(* Logix 5000 project; controller cal1632 1756-L62 rev 16.20; software revision 16.05; part 23 of 57 *)
(* tags used below, declared in another part *)
   FAULT : BOOL;
   HMI : BOOL;
   p01r09_pb_global_reset : BOOL;
   p19_ai_prs : REAL;
   p19_ai_tc01 : REAL;
   p19_ao_cv : REAL;
   p19_di_tc01_bo : BOOL;
   p19_di_tc02_bo : BOOL;
   p19_dint_to_hmi : DINT[16];
   p19_do_pump : BOOL;
   p19_param_pid2_ff : REAL;
   p19_param_pid2_kd : REAL;
   p19_param_pid2_ki : REAL;
   p19_param_pid2_kp : REAL;
   p19_param_tc01_dev : REAL;
   p19_param_tc01z : REAL;
   p19_param_tc02z : REAL;
   p19_param_zone_pressure : REAL;
   p19_real_to_hmi : REAL[80];
   p19r05 : routine;
   p19r05_timer_fault : TIMER[4];
   p19r05_timer_warning : TIMER[4];
   p19r06 : routine;
   p19r06_timer_fault : TIMER[4];
   p19r06_timer_warning : TIMER[4];
   p19r07 : routine;
   p19r07_timer_fault : TIMER[4];
   p19r07_timer_warning : TIMER[4];
   p19r30 : routine;
   p19r30_cv_man_sp : REAL;
   p19r30_pid_temp : PID;
   p19r30_pid_temp_pv : DINT;
   p19r30_request_cool : BOOL;
   p19r30_request_manual : BOOL;
   p19r31 : routine;
   p19r31_request_auto_run : BOOL;
(* P19_Advanced_Cooling, continued *)

ROUTINE R05_Dint_to_HMI   (* ladder *)
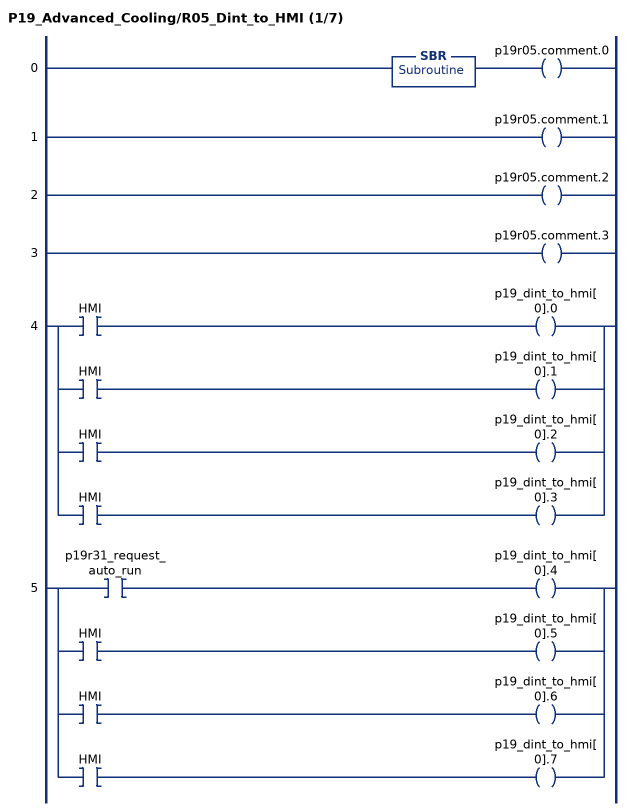
   0: SBR()OTE(p19r05.comment.0);
   1: OTE(p19r05.comment.1);
   2: OTE(p19r05.comment.2);
   3: OTE(p19r05.comment.3);
   4: [XIC(HMI) OTE(p19_dint_to_hmi[0].0) ,XIC(HMI) OTE(p19_dint_to_hmi[0].1) ,XIC(HMI) OTE(p19_dint_to_hmi[0].2) ,XIC(HMI) OTE(p19_dint_to_hmi[0].3) ];
   5: [XIC(p19r31_request_auto_run) OTE(p19_dint_to_hmi[0].4) ,XIC(HMI) OTE(p19_dint_to_hmi[0].5) ,XIC(HMI) OTE(p19_dint_to_hmi[0].6) ,XIC(HMI) OTE(p19_dint_to_hmi[0].7) ];
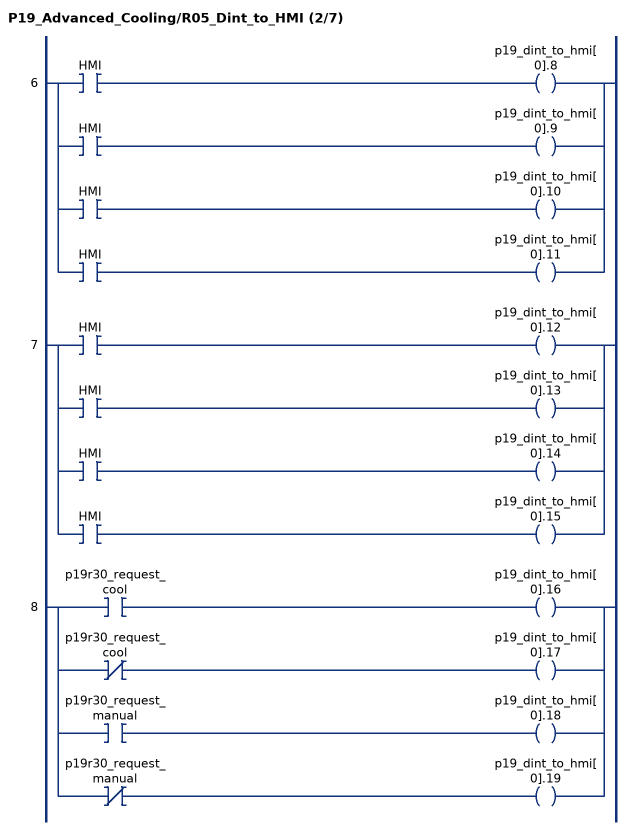
   6: [XIC(HMI) OTE(p19_dint_to_hmi[0].8) ,XIC(HMI) OTE(p19_dint_to_hmi[0].9) ,XIC(HMI) OTE(p19_dint_to_hmi[0].10) ,XIC(HMI) OTE(p19_dint_to_hmi[0].11) ];
   7: [XIC(HMI) OTE(p19_dint_to_hmi[0].12) ,XIC(HMI) OTE(p19_dint_to_hmi[0].13) ,XIC(HMI) OTE(p19_dint_to_hmi[0].14) ,XIC(HMI) OTE(p19_dint_to_hmi[0].15) ];
   8: [XIC(p19r30_request_cool) OTE(p19_dint_to_hmi[0].16) ,XIO(p19r30_request_cool) OTE(p19_dint_to_hmi[0].17) ,XIC(p19r30_request_manual) OTE(p19_dint_to_hmi[0].18) ,XIO(p19r30_request_manual) OTE(p19_dint_to_hmi[0].19) ];
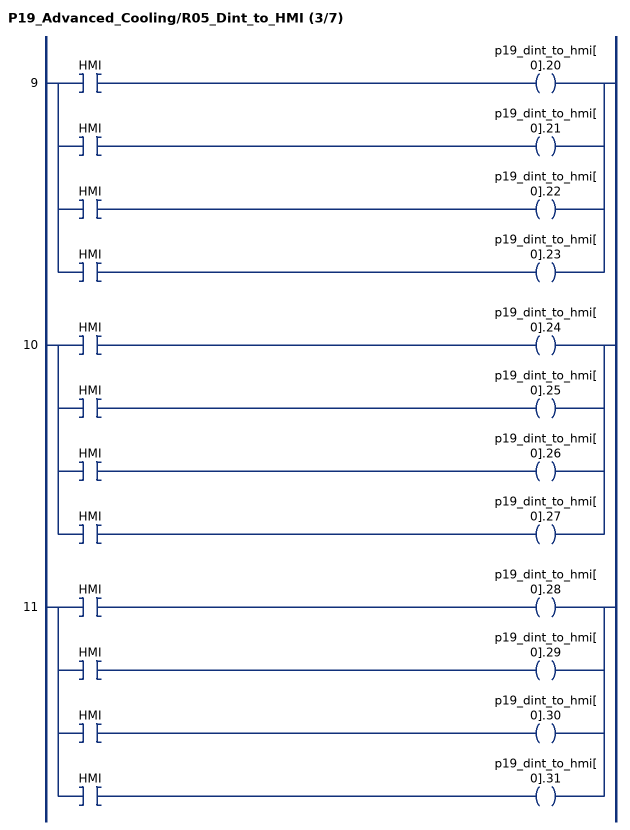
   9: [XIC(HMI) OTE(p19_dint_to_hmi[0].20) ,XIC(HMI) OTE(p19_dint_to_hmi[0].21) ,XIC(HMI) OTE(p19_dint_to_hmi[0].22) ,XIC(HMI) OTE(p19_dint_to_hmi[0].23) ];
   10: [XIC(HMI) OTE(p19_dint_to_hmi[0].24) ,XIC(HMI) OTE(p19_dint_to_hmi[0].25) ,XIC(HMI) OTE(p19_dint_to_hmi[0].26) ,XIC(HMI) OTE(p19_dint_to_hmi[0].27) ];
   11: [XIC(HMI) OTE(p19_dint_to_hmi[0].28) ,XIC(HMI) OTE(p19_dint_to_hmi[0].29) ,XIC(HMI) OTE(p19_dint_to_hmi[0].30) ,XIC(HMI) OTE(p19_dint_to_hmi[0].31) ];
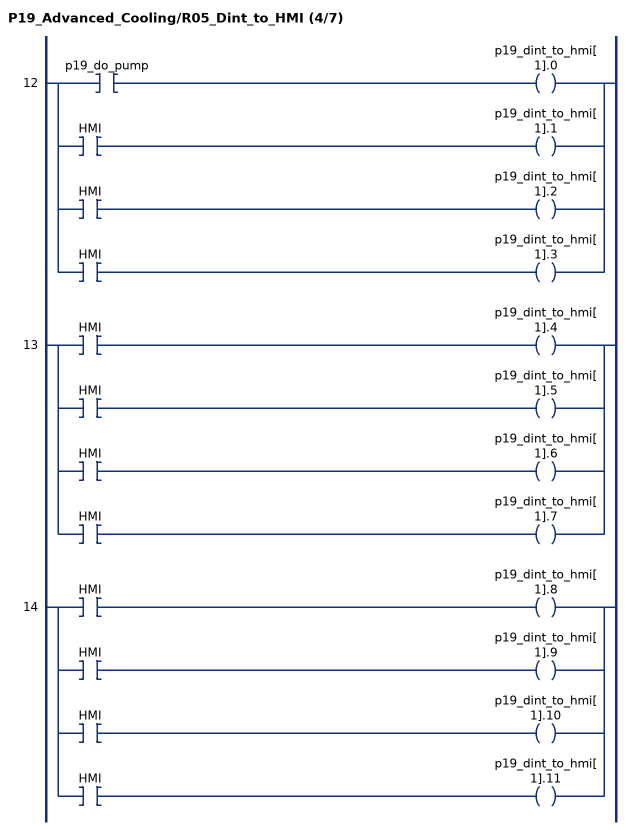
   12: [XIC(p19_do_pump) OTE(p19_dint_to_hmi[1].0) ,XIC(HMI) OTE(p19_dint_to_hmi[1].1) ,XIC(HMI) OTE(p19_dint_to_hmi[1].2) ,XIC(HMI) OTE(p19_dint_to_hmi[1].3) ];
   13: [XIC(HMI) OTE(p19_dint_to_hmi[1].4) ,XIC(HMI) OTE(p19_dint_to_hmi[1].5) ,XIC(HMI) OTE(p19_dint_to_hmi[1].6) ,XIC(HMI) OTE(p19_dint_to_hmi[1].7) ];
   14: [XIC(HMI) OTE(p19_dint_to_hmi[1].8) ,XIC(HMI) OTE(p19_dint_to_hmi[1].9) ,XIC(HMI) OTE(p19_dint_to_hmi[1].10) ,XIC(HMI) OTE(p19_dint_to_hmi[1].11) ];
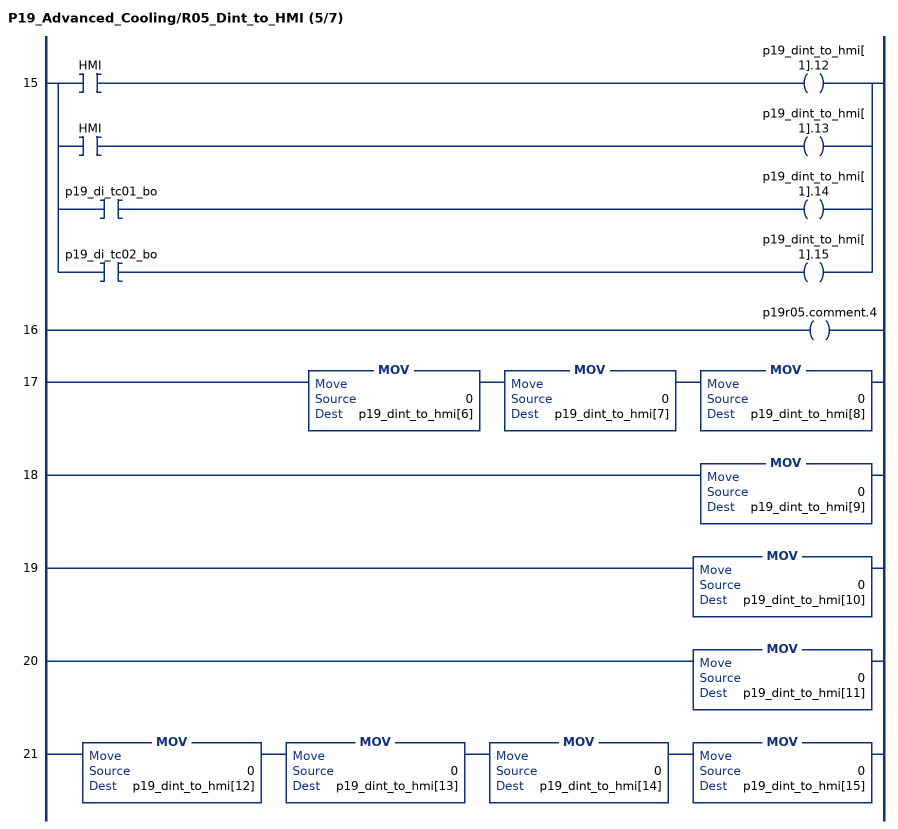
   15: [XIC(HMI) OTE(p19_dint_to_hmi[1].12) ,XIC(HMI) OTE(p19_dint_to_hmi[1].13) ,XIC(p19_di_tc01_bo) OTE(p19_dint_to_hmi[1].14) ,XIC(p19_di_tc02_bo) OTE(p19_dint_to_hmi[1].15) ];
   16: OTE(p19r05.comment.4);
   17: MOV(0,p19_dint_to_hmi[6])MOV(0,p19_dint_to_hmi[7])MOV(0,p19_dint_to_hmi[8]);
   18: MOV(0,p19_dint_to_hmi[9]);
   19: MOV(0,p19_dint_to_hmi[10]);
   20: MOV(0,p19_dint_to_hmi[11]);
   21: MOV(0,p19_dint_to_hmi[12])MOV(0,p19_dint_to_hmi[13])MOV(0,p19_dint_to_hmi[14])MOV(0,p19_dint_to_hmi[15]);
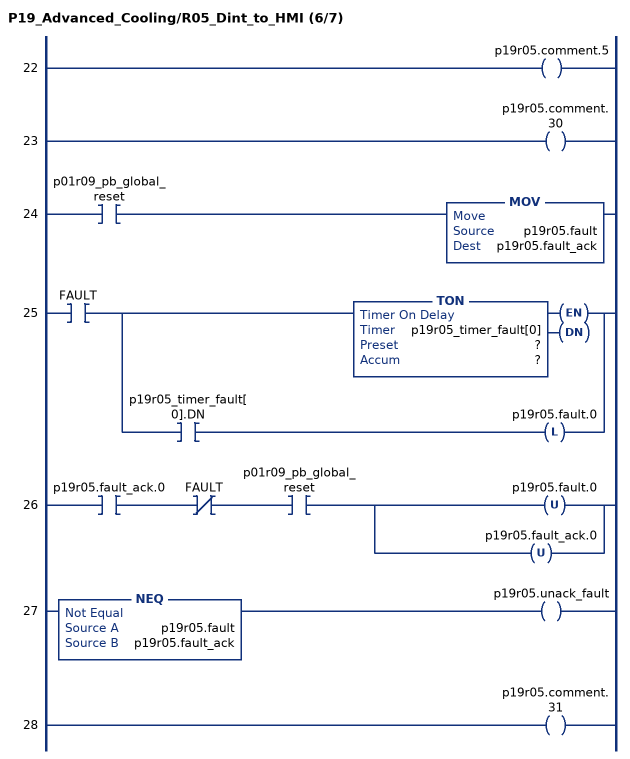
   22: OTE(p19r05.comment.5);
   23: OTE(p19r05.comment.30);
   24: XIC(p01r09_pb_global_reset)MOV(p19r05.fault,p19r05.fault_ack);
   25: XIC(FAULT)[TON(p19r05_timer_fault[0],?,?) ,XIC(p19r05_timer_fault[0].DN) OTL(p19r05.fault.0) ];
   26: XIC(p19r05.fault_ack.0)XIO(FAULT)XIC(p01r09_pb_global_reset)[OTU(p19r05.fault.0) ,OTU(p19r05.fault_ack.0) ];
   27: NEQ(p19r05.fault,p19r05.fault_ack)OTE(p19r05.unack_fault);
   28: OTE(p19r05.comment.31);
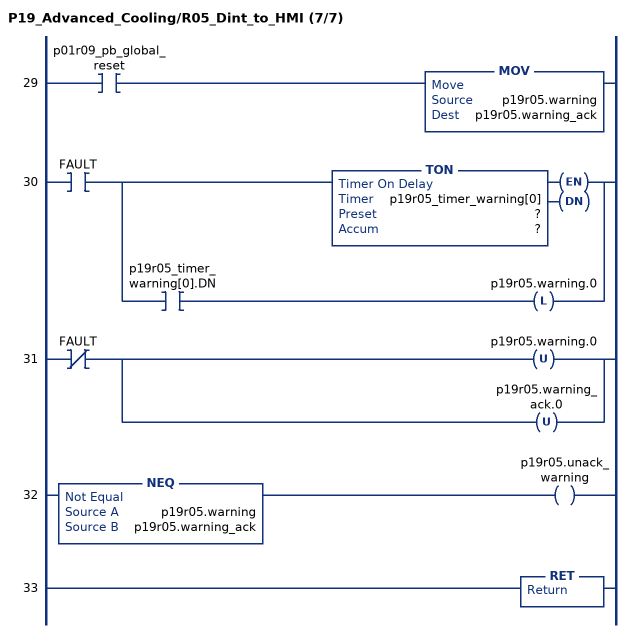
   29: XIC(p01r09_pb_global_reset)MOV(p19r05.warning,p19r05.warning_ack);
   30: XIC(FAULT)[TON(p19r05_timer_warning[0],?,?) ,XIC(p19r05_timer_warning[0].DN) OTL(p19r05.warning.0) ];
   31: XIO(FAULT)[OTU(p19r05.warning.0) ,OTU(p19r05.warning_ack.0) ];
   32: NEQ(p19r05.warning,p19r05.warning_ack)OTE(p19r05.unack_warning);
   33: RET();
END_ROUTINE

ROUTINE R06_Real_to_HMI   (* ladder *)
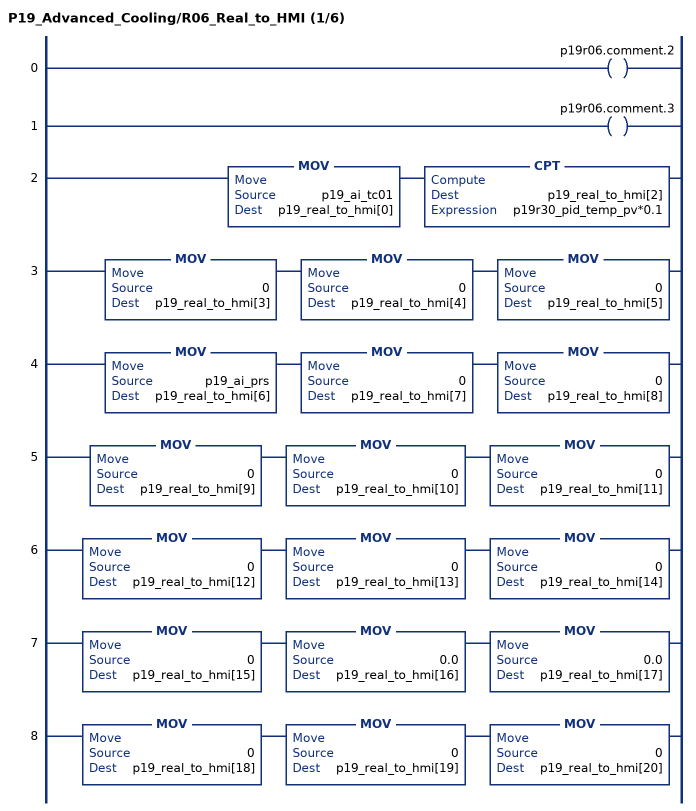
   0: OTE(p19r06.comment.2);
   1: OTE(p19r06.comment.3);
   2: MOV(p19_ai_tc01,p19_real_to_hmi[0])CPT(p19_real_to_hmi[2],p19r30_pid_temp_pv*0.1);
   3: MOV(0,p19_real_to_hmi[3])MOV(0,p19_real_to_hmi[4])MOV(0,p19_real_to_hmi[5]);
   4: MOV(p19_ai_prs,p19_real_to_hmi[6])MOV(0,p19_real_to_hmi[7])MOV(0,p19_real_to_hmi[8]);
   5: MOV(0,p19_real_to_hmi[9])MOV(0,p19_real_to_hmi[10])MOV(0,p19_real_to_hmi[11]);
   6: MOV(0,p19_real_to_hmi[12])MOV(0,p19_real_to_hmi[13])MOV(0,p19_real_to_hmi[14]);
   7: MOV(0,p19_real_to_hmi[15])MOV(0.0,p19_real_to_hmi[16])MOV(0.0,p19_real_to_hmi[17]);
   8: MOV(0,p19_real_to_hmi[18])MOV(0,p19_real_to_hmi[19])MOV(0,p19_real_to_hmi[20]);
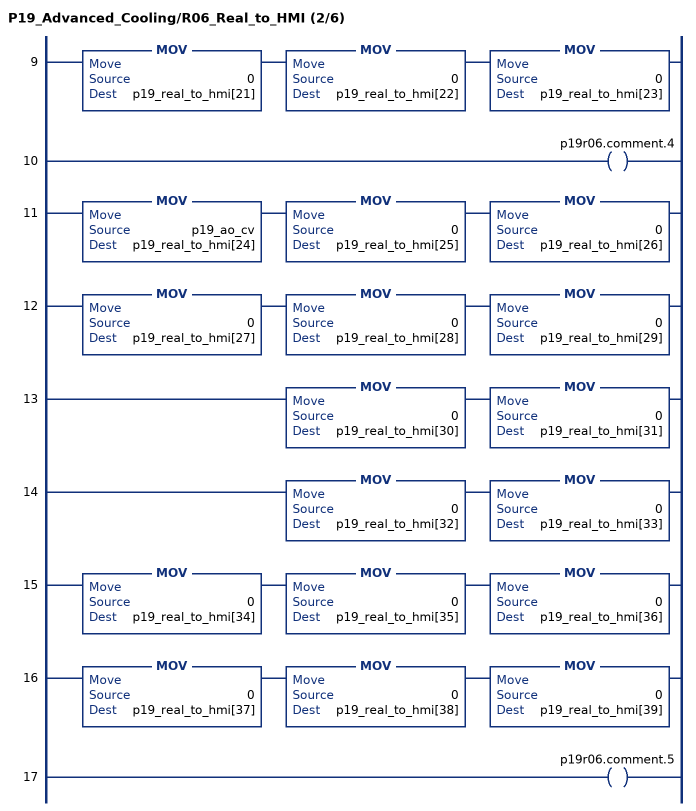
   9: MOV(0,p19_real_to_hmi[21])MOV(0,p19_real_to_hmi[22])MOV(0,p19_real_to_hmi[23]);
   10: OTE(p19r06.comment.4);
   11: MOV(p19_ao_cv,p19_real_to_hmi[24])MOV(0,p19_real_to_hmi[25])MOV(0,p19_real_to_hmi[26]);
   12: MOV(0,p19_real_to_hmi[27])MOV(0,p19_real_to_hmi[28])MOV(0,p19_real_to_hmi[29]);
   13: MOV(0,p19_real_to_hmi[30])MOV(0,p19_real_to_hmi[31]);
   14: MOV(0,p19_real_to_hmi[32])MOV(0,p19_real_to_hmi[33]);
   15: MOV(0,p19_real_to_hmi[34])MOV(0,p19_real_to_hmi[35])MOV(0,p19_real_to_hmi[36]);
   16: MOV(0,p19_real_to_hmi[37])MOV(0,p19_real_to_hmi[38])MOV(0,p19_real_to_hmi[39]);
   17: OTE(p19r06.comment.5);
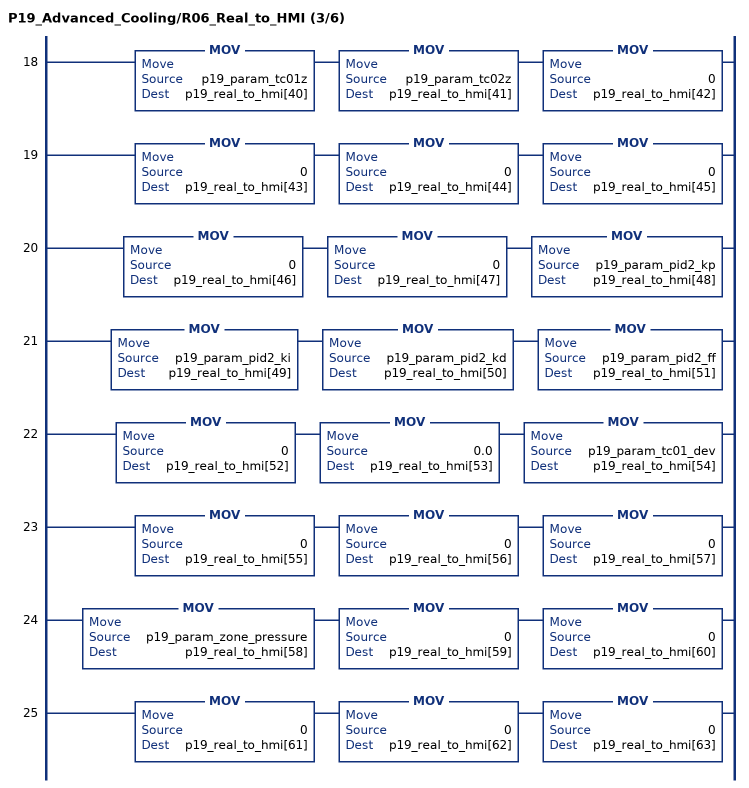
   18: MOV(p19_param_tc01z,p19_real_to_hmi[40])MOV(p19_param_tc02z,p19_real_to_hmi[41])MOV(0,p19_real_to_hmi[42]);
   19: MOV(0,p19_real_to_hmi[43])MOV(0,p19_real_to_hmi[44])MOV(0,p19_real_to_hmi[45]);
   20: MOV(0,p19_real_to_hmi[46])MOV(0,p19_real_to_hmi[47])MOV(p19_param_pid2_kp,p19_real_to_hmi[48]);
   21: MOV(p19_param_pid2_ki,p19_real_to_hmi[49])MOV(p19_param_pid2_kd,p19_real_to_hmi[50])MOV(p19_param_pid2_ff,p19_real_to_hmi[51]);
   22: MOV(0,p19_real_to_hmi[52])MOV(0.0,p19_real_to_hmi[53])MOV(p19_param_tc01_dev,p19_real_to_hmi[54]);
   23: MOV(0,p19_real_to_hmi[55])MOV(0,p19_real_to_hmi[56])MOV(0,p19_real_to_hmi[57]);
   24: MOV(p19_param_zone_pressure,p19_real_to_hmi[58])MOV(0,p19_real_to_hmi[59])MOV(0,p19_real_to_hmi[60]);
   25: MOV(0,p19_real_to_hmi[61])MOV(0,p19_real_to_hmi[62])MOV(0,p19_real_to_hmi[63]);
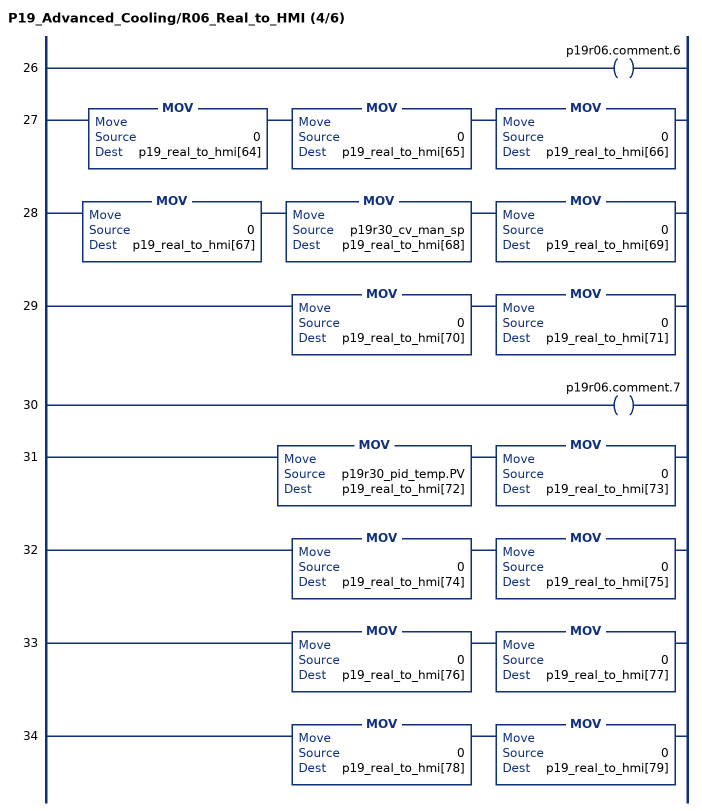
   26: OTE(p19r06.comment.6);
   27: MOV(0,p19_real_to_hmi[64])MOV(0,p19_real_to_hmi[65])MOV(0,p19_real_to_hmi[66]);
   28: MOV(0,p19_real_to_hmi[67])MOV(p19r30_cv_man_sp,p19_real_to_hmi[68])MOV(0,p19_real_to_hmi[69]);
   29: MOV(0,p19_real_to_hmi[70])MOV(0,p19_real_to_hmi[71]);
   30: OTE(p19r06.comment.7);
   31: MOV(p19r30_pid_temp.PV,p19_real_to_hmi[72])MOV(0,p19_real_to_hmi[73]);
   32: MOV(0,p19_real_to_hmi[74])MOV(0,p19_real_to_hmi[75]);
   33: MOV(0,p19_real_to_hmi[76])MOV(0,p19_real_to_hmi[77]);
   34: MOV(0,p19_real_to_hmi[78])MOV(0,p19_real_to_hmi[79]);
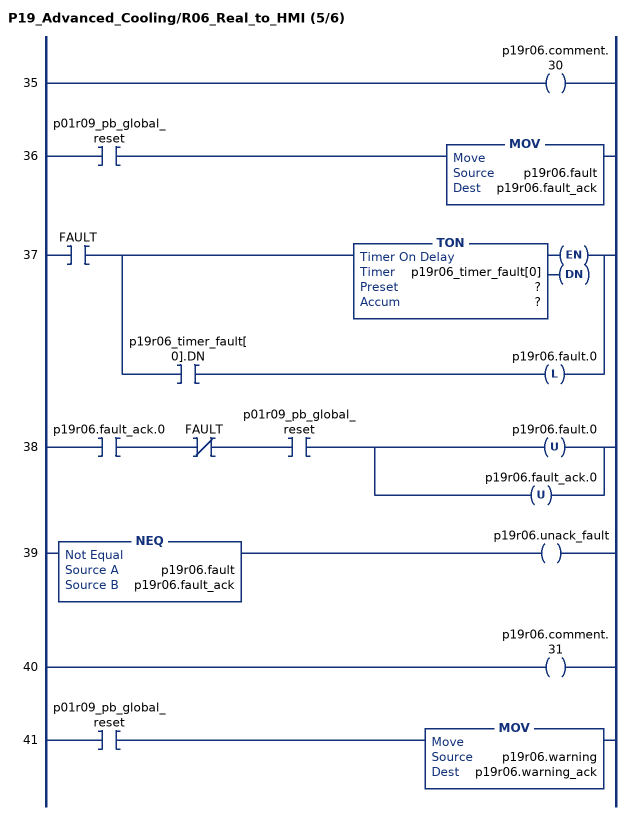
   35: OTE(p19r06.comment.30);
   36: XIC(p01r09_pb_global_reset)MOV(p19r06.fault,p19r06.fault_ack);
   37: XIC(FAULT)[TON(p19r06_timer_fault[0],?,?) ,XIC(p19r06_timer_fault[0].DN) OTL(p19r06.fault.0) ];
   38: XIC(p19r06.fault_ack.0)XIO(FAULT)XIC(p01r09_pb_global_reset)[OTU(p19r06.fault.0) ,OTU(p19r06.fault_ack.0) ];
   39: NEQ(p19r06.fault,p19r06.fault_ack)OTE(p19r06.unack_fault);
   40: OTE(p19r06.comment.31);
   41: XIC(p01r09_pb_global_reset)MOV(p19r06.warning,p19r06.warning_ack);
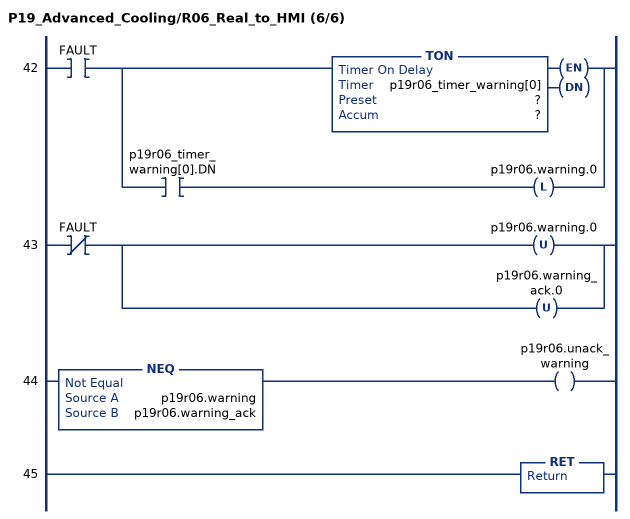
   42: XIC(FAULT)[TON(p19r06_timer_warning[0],?,?) ,XIC(p19r06_timer_warning[0].DN) OTL(p19r06.warning.0) ];
   43: XIO(FAULT)[OTU(p19r06.warning.0) ,OTU(p19r06.warning_ack.0) ];
   44: NEQ(p19r06.warning,p19r06.warning_ack)OTE(p19r06.unack_warning);
   45: RET();
END_ROUTINE

ROUTINE R07_Alarms   (* ladder *)
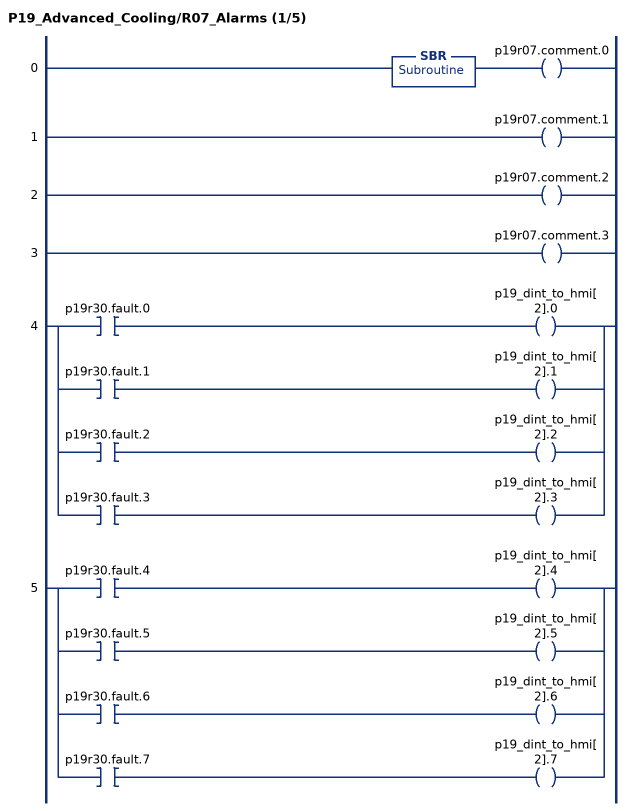
   0: SBR()OTE(p19r07.comment.0);
   1: OTE(p19r07.comment.1);
   2: OTE(p19r07.comment.2);
   3: OTE(p19r07.comment.3);
   4: [XIC(p19r30.fault.0) OTE(p19_dint_to_hmi[2].0) ,XIC(p19r30.fault.1) OTE(p19_dint_to_hmi[2].1) ,XIC(p19r30.fault.2) OTE(p19_dint_to_hmi[2].2) ,XIC(p19r30.fault.3) OTE(p19_dint_to_hmi[2].3) ];
   5: [XIC(p19r30.fault.4) OTE(p19_dint_to_hmi[2].4) ,XIC(p19r30.fault.5) OTE(p19_dint_to_hmi[2].5) ,XIC(p19r30.fault.6) OTE(p19_dint_to_hmi[2].6) ,XIC(p19r30.fault.7) OTE(p19_dint_to_hmi[2].7) ];
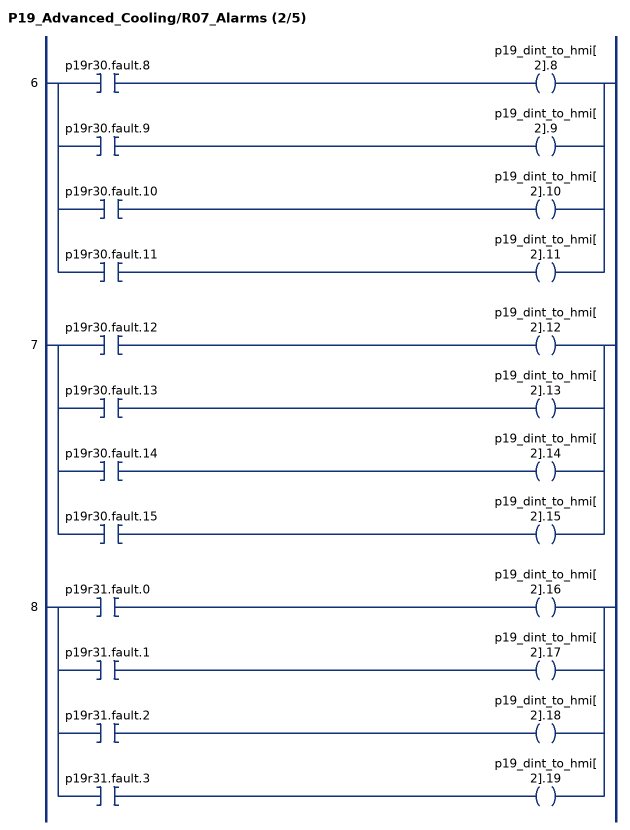
   6: [XIC(p19r30.fault.8) OTE(p19_dint_to_hmi[2].8) ,XIC(p19r30.fault.9) OTE(p19_dint_to_hmi[2].9) ,XIC(p19r30.fault.10) OTE(p19_dint_to_hmi[2].10) ,XIC(p19r30.fault.11) OTE(p19_dint_to_hmi[2].11) ];
   7: [XIC(p19r30.fault.12) OTE(p19_dint_to_hmi[2].12) ,XIC(p19r30.fault.13) OTE(p19_dint_to_hmi[2].13) ,XIC(p19r30.fault.14) OTE(p19_dint_to_hmi[2].14) ,XIC(p19r30.fault.15) OTE(p19_dint_to_hmi[2].15) ];
   8: [XIC(p19r31.fault.0) OTE(p19_dint_to_hmi[2].16) ,XIC(p19r31.fault.1) OTE(p19_dint_to_hmi[2].17) ,XIC(p19r31.fault.2) OTE(p19_dint_to_hmi[2].18) ,XIC(p19r31.fault.3) OTE(p19_dint_to_hmi[2].19) ];
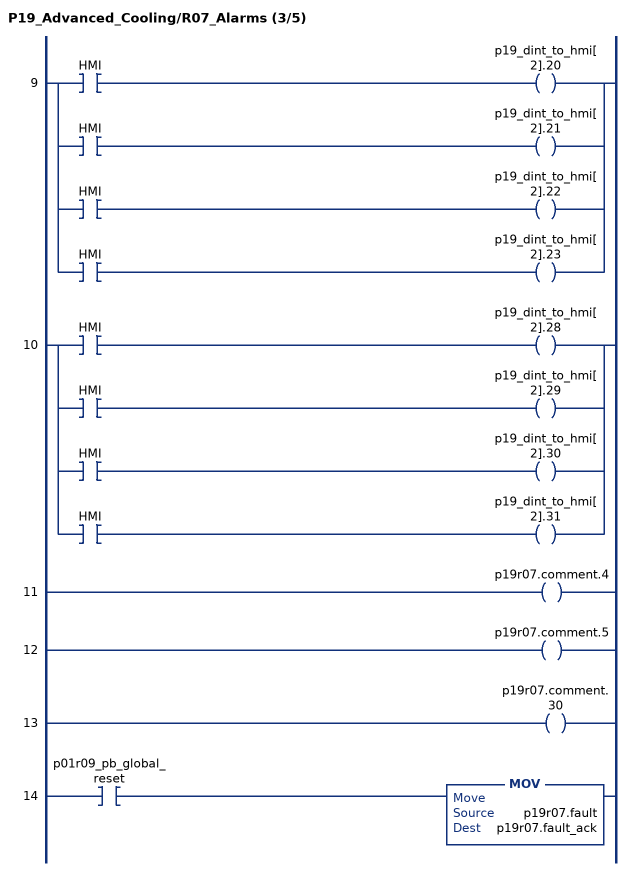
   9: [XIC(HMI) OTE(p19_dint_to_hmi[2].20) ,XIC(HMI) OTE(p19_dint_to_hmi[2].21) ,XIC(HMI) OTE(p19_dint_to_hmi[2].22) ,XIC(HMI) OTE(p19_dint_to_hmi[2].23) ];
   10: [XIC(HMI) OTE(p19_dint_to_hmi[2].28) ,XIC(HMI) OTE(p19_dint_to_hmi[2].29) ,XIC(HMI) OTE(p19_dint_to_hmi[2].30) ,XIC(HMI) OTE(p19_dint_to_hmi[2].31) ];
   11: OTE(p19r07.comment.4);
   12: OTE(p19r07.comment.5);
   13: OTE(p19r07.comment.30);
   14: XIC(p01r09_pb_global_reset)MOV(p19r07.fault,p19r07.fault_ack);
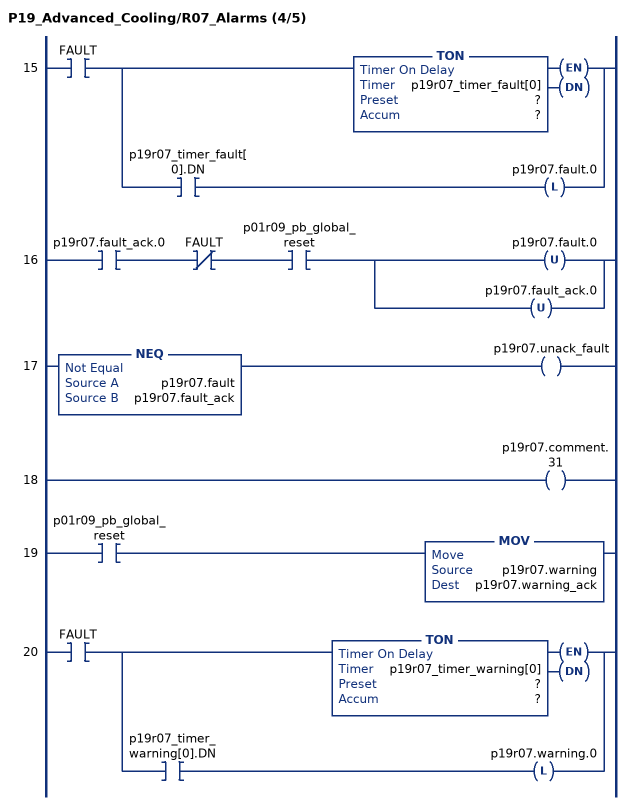
   15: XIC(FAULT)[TON(p19r07_timer_fault[0],?,?) ,XIC(p19r07_timer_fault[0].DN) OTL(p19r07.fault.0) ];
   16: XIC(p19r07.fault_ack.0)XIO(FAULT)XIC(p01r09_pb_global_reset)[OTU(p19r07.fault.0) ,OTU(p19r07.fault_ack.0) ];
   17: NEQ(p19r07.fault,p19r07.fault_ack)OTE(p19r07.unack_fault);
   18: OTE(p19r07.comment.31);
   19: XIC(p01r09_pb_global_reset)MOV(p19r07.warning,p19r07.warning_ack);
   20: XIC(FAULT)[TON(p19r07_timer_warning[0],?,?) ,XIC(p19r07_timer_warning[0].DN) OTL(p19r07.warning.0) ];
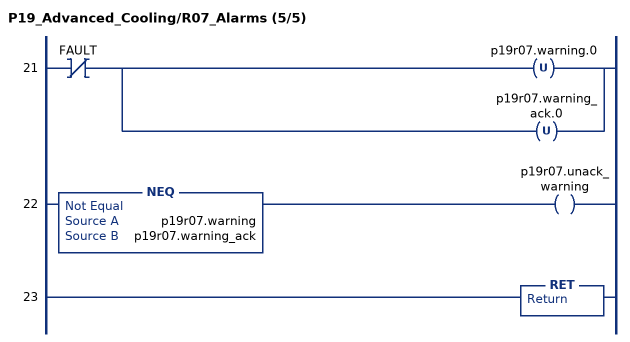
   21: XIO(FAULT)[OTU(p19r07.warning.0) ,OTU(p19r07.warning_ack.0) ];
   22: NEQ(p19r07.warning,p19r07.warning_ack)OTE(p19r07.unack_warning);
   23: RET();
END_ROUTINE
